{attribute 'linkalways'} 
{attribute 'no_explicit_call' := 'This FB is a CLASS and must be accessed using methods or properties'}
{attribute 'enable_dynamic_creation'}
FUNCTION_BLOCK _ETcVnRotationAngle EXTENDS EnumDatatypeBase
VAR
	localData : ETcVnRotationAngle;
	activeData : REFERENCE TO ETcVnRotationAngle;
	enumBaseDatatype : _DINT(localData);
END_VAR

METHOD PRIVATE AddLocalEnumeration
VAR_INPUT
	Enumeration : T_MAXSTRING;
	Value : ETcVnRotationAngle;
END_VAR
AddEnumeration(Enumeration, Value);
END_METHOD

PROPERTY PUBLIC Address : PVOID
GET
Address := ADR(activeData);
END_GET
END_PROPERTY

METHOD PUBLIC ClearReference
VAR_INPUT
END_VAR
activeData REF= localData;
SetBaseDatatypeReference();
END_METHOD

METHOD PUBLIC Clone : I_Datatype
VAR
    pClone : POINTER TO _ETcVnRotationAngle;
END_VAR
pClone := __NEW(_ETcVnRotationAngle(InitialValue := Value));
Clone := pClone^;
END_METHOD

METHOD FB_init : BOOL
VAR_INPUT
	bInitRetains : BOOL; // if TRUE, the retain variables are initialized (warm start / cold start)
	bInCopyCode : BOOL;  // if TRUE, the instance afterwards gets moved into the copy code (online change)
	InitialValue : ETcVnRotationAngle;
END_VAR
localData := InitialValue;
AddBaseDatatype(enumBaseDatatype);
ClearReference();

AddLocalEnumeration('TCVN_RA_90_DEG', ETcVnRotationAngle.TCVN_RA_90_DEG);
AddLocalEnumeration('TCVN_RA_180_DEG', ETcVnRotationAngle.TCVN_RA_180_DEG);
AddLocalEnumeration('TCVN_RA_270_DEG', ETcVnRotationAngle.TCVN_RA_270_DEG);
END_METHOD

PROPERTY PUBLIC Identifier : T_MAXSTRING
GET
Identifier := 'ETcVnRotationAngle';
END_GET
END_PROPERTY

METHOD IsEnumeratorValueEqual : BOOL
VAR_INPUT
	Enumerator : I_KeyValueForwardEnumerator;
END_VAR
VAR
	storedValue : ETcVnRotationAngle;
END_VAR
IF NOT Enumerator.TryGet(storedValue) THEN
	RETURN;
END_IF

IsEnumeratorValueEqual := storedValue = activeData;
END_METHOD

METHOD PUBLIC MakeReferenceTo
VAR_INPUT
	ReferenceTarget : REFERENCE TO ETcVnRotationAngle;
END_VAR
activeData REF= ReferenceTarget;
SetBaseDatatypeReference();
END_METHOD

METHOD PROTECTED SetBaseDatatypeReference
VAR_INPUT
END_VAR
enumBaseDatatype.MakeReferenceTo(activeData);
END_METHOD

PROPERTY PUBLIC Size : UDINT
GET
Size := SIZEOF(activeData);
END_GET
END_PROPERTY

METHOD TryMakeReferenceTo : BOOL
VAR_INPUT
	Target : I_Datatype;
END_VAR
VAR
	pTargetData : POINTER TO ETcVnRotationAngle;
END_VAR
IF NOT IsEquivalentTo(Target) THEN
	RETURN;
END_IF

pTargetData := Target.Address;
activeData REF= pTargetData^;
SetBaseDatatypeReference();
TryMakeReferenceTo := TRUE;
END_METHOD

PROPERTY PUBLIC Value : ETcVnRotationAngle
GET
Value := activeData;
END_GET
SET
activeData := Value;
END_SET
END_PROPERTY

END_FUNCTION_BLOCK

(* stored: Version 1.1.0.1, ProductVersion 3.1.4024.13
   POU _ETcVnRotationAngle: Id {3ed53119-6131-0e45-0271-e93f9cd42ebe}, SpecialFunc None
   Folder Core: Id {429172dd-71f1-0427-3620-2c52bf54c7f5}
   Folder Protected: Id {be7ac666-32a2-0123-1434-1e0985e8c513}
   Folder Customize: Id {4fa9d402-8932-0179-1246-73fe94db4254}
   Folder Constructor: Id {59ef69ae-3a1c-0a21-0b47-e48af5bf9a9c}
   Folder Private: Id {a31acba8-c4f0-0fd2-2f11-ff283cff551f}
   Folder Protected: Id {e115d151-605f-058e-2cb8-50ed6764f946}
   Method AddLocalEnumeration: Id {e2bbbff8-f3b9-0397-3f08-13e519fa54b2}
   Property Address: Id {96e8963f-35b9-06c7-03ce-0bb481cbcefd}
   Get Get: Id {fc772da6-fb7b-0a41-1ca2-6d33195847f9}
   Method ClearReference: Id {5d7e0c14-2fb9-07a3-0021-2953e9dff34b}
   Method Clone: Id {08dc178c-53ef-05f1-189a-41abd13f152b}
   Method FB_init: Id {650a1875-efe0-038e-1bc2-054636b2f7e0}
   Property Identifier: Id {d74d8cc5-9ad5-077b-05bd-9eb82e478536}
   Get Get: Id {52cfaf12-d690-0877-39b6-686f48bddfe8}
   Method IsEnumeratorValueEqual: Id {ede25439-f05d-0299-2927-8c9027810160}
   Method MakeReferenceTo: Id {2f738397-bde0-01dc-058b-7da9603e5e10}
   Method SetBaseDatatypeReference: Id {9b01c3da-9040-0e73-2811-ddeb5ac68c87}
   Property Size: Id {a5b00ec7-d764-09e2-0fd6-489d42e18ce8}
   Get Get: Id {31668984-74fa-0122-39fc-0d53c000a016}
   Method TryMakeReferenceTo: Id {297cbceb-8adf-0163-2024-37f5772b60ac}
   Property Value: Id {d23ab667-2de3-059b-1619-7c68a303157e}
   Get Get: Id {cc883cec-7edc-0af6-3866-304e1c37b3d8}
   Set Set: Id {9b457fac-c6ff-0287-1581-0ab7b3c4bf38} *)
